Universal Robots PolyScope program: _adminCG-InvDToPHome.urp

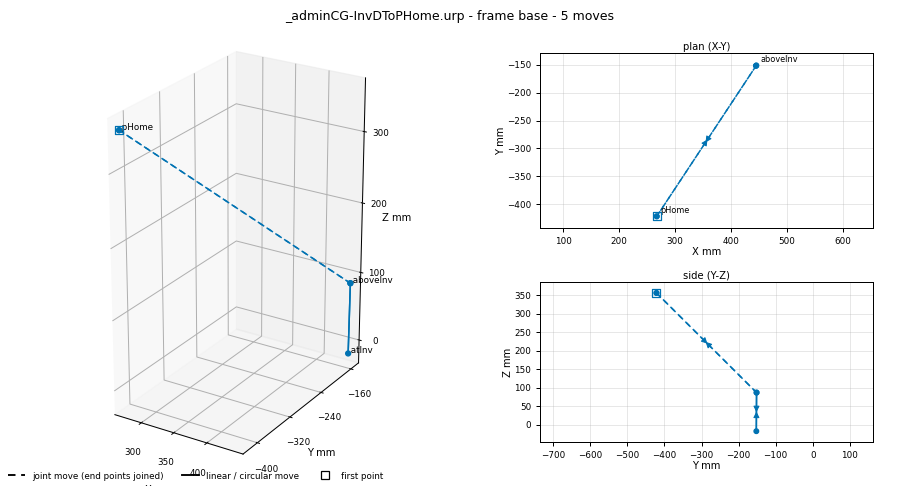
[picture p0: tool path of _adminCG-InvDToPHome.urp in frame base, 5 of 5 moves have a stored position in this frame; points joined in program order, loops and branches not executed]
Program _adminCG-InvDToPHome (installation=admin directory=/programs/THU_530PM createdIn=3.8.0.61336 lastSavedIn=3.15.8.106339 robotSerialNumber=2015350924)
Calibrated DH parameters: a=[0, -0.425, -0.39225, 0, 0, 0]; d=[0.089159, 0, 0, 0.10915, 0.09465, 0.0823]; alpha=[1.570796, 0, 0, 1.570796, -1.570796, 0]; deltaTheta=[0, 0, 0, 0, 0, 0]
Robot Program (runOnlyOnce=true)
  Set DigitalOutput pin=digital_out[0]; digitalValue=0
  Call _adminLinearIndex4
  MoveJ speed 60 deg/s, acceleration 80 deg/s^2 (useActiveTCP=true)
    Waypoint pHome: TCP in base x=267.077 y=-421.526 z=355.862 mm, rx=1.114 ry=1.1061 rz=0.0051 rad; joints [-45.007, -90.005, -89.993, -90.005, 90, -0.004] deg; flange x=267.08 y=-421.53 z=431.862 mm, rx=1.2021 ry=-2.9025 rz=-0.0001 rad
    Waypoint aboveInv: TCP in base x=445.29 y=-151.53 z=87.176 mm, rx=1.1162 ry=1.1066 rz=-0.0013 rad; joints [-5.351, -99.714, -122.242, -48.254, 89.929, 39.928] deg; flange x=445.577 y=-151.462 z=163.175 mm, rx=1.1937 ry=-2.9018 rz=-0.0009 rad
  MoveL speed 250 mm/s, acceleration 1200 mm/s^2 (useActiveTCP=true) feature=Base
    Waypoint atInv: TCP in base x=444.627 y=-152.161 z=-16.997 mm, rx=1.1162 ry=1.1067 rz=-0.0013 rad; joints [-5.437, -112.925, -126.853, -30.436, 89.929, 39.841] deg; flange x=444.918 y=-152.094 z=59.002 mm, rx=1.1937 ry=-2.9018 rz=-0.001 rad
    Set DigitalOutput pin=digital_out[0]; digitalValue=1
    Wait Sleep waitTime=1
    Waypoint aboveInv: TCP in base x=445.29 y=-151.53 z=87.176 mm, rx=1.1162 ry=1.1066 rz=-0.0013 rad; joints [-5.351, -99.714, -122.242, -48.254, 89.929, 39.928] deg; flange x=445.577 y=-151.462 z=163.175 mm, rx=1.1937 ry=-2.9018 rz=-0.0009 rad
  MoveJ speed 180 deg/s, acceleration 100 deg/s^2 (useActiveTCP=true)
    Waypoint phome: TCP in base x=267.106 y=-421.453 z=355.828 mm, rx=1.114 ry=1.1062 rz=0.0052 rad; joints [-45, -90.001, -90.002, -90.005, 90.003, -0.002] deg; flange x=267.11 y=-421.463 z=431.828 mm, rx=1.2023 ry=-2.9024 rz=-0.0002 rad
SubProgram  [hidden by the author, left out]
SubProgram _adminLinearIndex4 [hidden by the author, left out]
